// Mitsubishi GX Works2 project: 闪烁八次后常亮   PLC: FX1S

PROGRAM MAIN
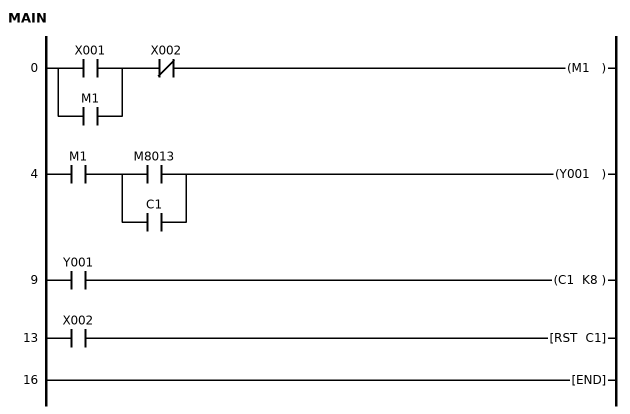
0     LD      X001
      OR      M1
      ANI     X002
      OUT     M1
4     LD      M1
      LD      M8013
      OR      C1
      ANB
      OUT     Y001
9     LD      Y001
      OUT     C1 K8
13    LD      X002
      RST     C1
16    END
END_PROGRAM
